PROGRAM MAIN
VAR
END_VAR

END_PROGRAM

(* stored: Version 1.1.0.1
   POU MAIN: Id {4d888670-415c-439f-8192-7f3914a5ea31} *)
